(* PLC project  *)

PROGRAM P

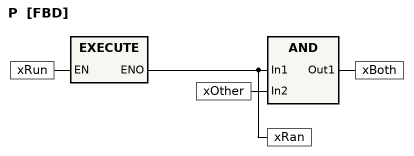
(* FBD diagram, written out as Structured Text *)
IF xRun THEN
  nCount := nCount + 1;
END_IF;
xRan := xRun;
xBoth := xRun AND xOther;
END_PROGRAM
